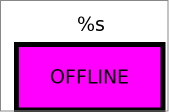
VISUALIZATION Obj_PDU_Surge  // 169x112
VAR_INPUT
	sIndex : STRING;
	bAlarm : BOOL;
	bOffline : BOOL;
END_VAR
    Rectangle (14,42 151x70), "%s", colour toggle: bAlarm, text list: 'PDU_Surge_Status', text index: bAlarm
    Rectangle (14,42 151x70), "OFFLINE", invisible if: not bOffline
    Rectangle (13,6 156x37), "%s", text variable: sIndex
END_VISUALIZATION

(* stored: Version 1.1.0.1, ProductVersion 3.1.4024.12
   Visu Obj_PDU_Surge: Id {6368e2b2-962a-4c43-acda-9cdad73b17ea} *)
